Universal Robots PolyScope program: lift column test.urp

Program lift column test (installation=default directory=/programs createdIn=5.14.5 lastSavedIn=5.14.5 robotSerialNumber=20236801216)
Calibrated DH parameters: a=[-0.000021, -0.748897, -0.28186, -0.00004, -0.000055, 0]; d=[0.236225, -424.082933, -1564.66872, 1988.95162, 0.159094, 0.153873]; alpha=[1.570844, 0.001002, 0.000337, 1.571488, -1.569996, 0]; deltaTheta=[0, -0.516316, 5.626292, 1.173211, 0.000001, 0]
InitVariablesNode
Robot Program (runOnlyOnce=true)
  Wait Sleep waitTime=5
  'send up'
  URCap MachineLogic for Universal Robots (MachineLogic for Universal Robots, Vention Inc.) dataModel(numberAdded=0, acceleration_in_mm_per_s2=50.0, ActuatorPos=868.7, type=addMotor, teachColor=BLUE, combo1=MachineMotion1, combo2=(1) Custom Actuator, combo3=Move Relative, combo6=In series, message=Move Rel., description=Moves the actuator away from its current position by a given distance., comboAddress=Address 1, comboActuator=Valve 1, speed_in_mm_per_min=2400.0)
  Wait Sleep waitTime=5
  'send down'
  URCap MachineLogic for Universal Robots (MachineLogic for Universal Robots, Vention Inc.) dataModel(numberAdded=0, acceleration_in_mm_per_s2=50.0, type=addMotor, ActuatorPos=-868.7, teachColor=BLUE, combo1=MachineMotion1, combo2=(1) Custom Actuator, combo3=Move Relative, combo6=In series, message=Move Rel., description=Moves the actuator away from its current position by a given distance., comboAddress=Address 1, comboActuator=Valve 1, speed_in_mm_per_min=2400.0)
  Wait Sleep waitTime=5
